# Funcion para actualizar el color de la pieza
def actualizar_color(step_index, total_steps):
    factor = step_index / (total_steps - 1)
    rojo  = color_inicial[0] + (color_final[0] - color_inicial[0]) * factor
    verde = color_inicial[1] + (color_final[1] - color_inicial[1]) * factor
    azul  = color_inicial[2] + (color_final[2] - color_inicial[2]) * factor
    obj.setColor([rojo, verde, azul, 1.0])

for target_name in targets:
    target = RDK.Item(target_name, ITEM_TYPE_TARGET)
    if not target.Valid():
        raise Exception(f'Target no encontrado: {target_name}')
    target_poses.append(target.Pose())

total_steps = len(target_poses)

# Ir a posición de inicio
home_joints = robot.JointsHome()
robot.MoveJ(home_joints)
robot.MoveJ(target_poses[0])

RDK.Spray_SetState(SPRAY_ON)

# Pintado con cambio progresivo de color (10 pasos)
for i, pose in enumerate(target_poses[1:10]):

    actualizar_color(step_index, total_steps)
    robot.MoveL(pose)
    step_index += 1

# Últimos movimientos
robot.setSpeed(50, 50)
robot.setAcceleration(50)
actualizar_color(step_index, total_steps)
robot.MoveL(target_poses[10])
step_index += 1
actualizar_color(step_index, total_steps)
robot.MoveL(target_poses[11])
step_index += 1

robot.setSpeed(10, 10)
robot.setAcceleration(10)
for pose in target_poses[12:15]:
    actualizar_color(step_index, total_steps)
    robot.MoveJ(pose)
    step_index += 1

# Bucle: 18 pasos de 5 grados
for i in range(18):
    # Obtener la pose actual en cada iteración (actualizada)
    pose_actual6 = frame6.Pose()
    pose_actual5 = frame5.Pose()

    # Crear una rotación de 5 grados en Z
    rot_5deg6 = robomath.rotz(math.radians(5))
    rot_5deg5 = robomath.rotz(math.radians(5))

    # Aplicar rotación acumulativa
    nueva_pose6 = pose_actual6 * rot_5deg6
    nueva_pose5 = pose_actual5 * rot_5deg5

    # Establecer la nueva pose
    frame6.setPose(nueva_pose6)
    frame5.setPose(nueva_pose5)

for pose in target_poses[15:29]:
    actualizar_color(step_index, total_steps)
    robot.MoveJ(pose)
    step_index += 1

robot.MoveJ(home_joints)

for pose in target_poses[30:33]:
    actualizar_color(step_index, total_steps)
    robot.MoveJ(pose)
    step_index += 1

# Bucle: 18 pasos de 5 grados
for i in range(18):
    # Obtener la pose actual en cada iteración (actualizada)
    pose_actual6 = frame6.Pose()
    pose_actual5 = frame5.Pose()

    # Crear una rotación de 5 grados en Z
    rot_5deg6 = robomath.rotz(math.radians(5))
    rot_5deg5 = robomath.rotz(math.radians(5))

    # Aplicar rotación acumulativa
    nueva_pose6 = pose_actual6 * rot_5deg6
    nueva_pose5 = pose_actual5 * rot_5deg5

    # Establecer la nueva pose
    frame6.setPose(nueva_pose6)
    frame5.setPose(nueva_pose5)

for pose in target_poses[33:47]:
    actualizar_color(step_index, total_steps)
    robot.MoveJ(pose)
    step_index += 1

# Bucle: 18 pasos de 5 grados
for i in range(18):
    # Obtener la pose actual en cada iteración (actualizada)
    pose_actual6 = frame6.Pose()
    pose_actual5 = frame5.Pose()

    # Crear una rotación de 5 grados en Z
    rot_5deg6 = robomath.rotz(math.radians(5))
    rot_5deg5 = robomath.rotz(math.radians(5))

    # Aplicar rotación acumulativa
    nueva_pose6 = pose_actual6 * rot_5deg6
    nueva_pose5 = pose_actual5 * rot_5deg5

    # Establecer la nueva pose
    frame6.setPose(nueva_pose6)
    frame5.setPose(nueva_pose5)

for pose in target_poses[47:]:
    actualizar_color(step_index, total_steps)
    robot.MoveJ(pose)
    step_index += 1

# Bucle: 18 pasos de 5 grados
for i in range(18):
    # Obtener la pose actual en cada iteración (actualizada)
    pose_actual6 = frame6.Pose()
    pose_actual5 = frame5.Pose()

    # Crear una rotación de 5 grados en Z
    rot_5deg6 = robomath.rotz(math.radians(5))
    rot_5deg5 = robomath.rotz(math.radians(5))

    # Aplicar rotación acumulativa
    nueva_pose6 = pose_actual6 * rot_5deg6
    nueva_pose5 = pose_actual5 * rot_5deg5

    # Establecer la nueva pose
    frame6.setPose(nueva_pose6)
    frame5.setPose(nueva_pose5)

robot.MoveJ(home_joints)
time.sleep(5.0)

robot.MoveJ(home_joints)
robot.MoveJ(target_poses[0])

RDK.Spray_SetState(SPRAY_ON)

# Pintado con cambio progresivo de color (10 pasos)
for i, pose in enumerate(target_poses[1:10]):

    actualizar_color(step_index, total_steps)
    robot.MoveL(pose)
    step_index += 1

# Últimos movimientos
robot.setSpeed(50, 50)
robot.setAcceleration(50)
actualizar_color(step_index, total_steps)
robot.MoveL(target_poses[10])
step_index += 1
actualizar_color(step_index, total_steps)
robot.MoveL(target_poses[11])
step_index += 1

robot.setSpeed(10, 10)
robot.setAcceleration(10)
for pose in target_poses[12:15]:
    actualizar_color(step_index, total_steps)
    robot.MoveJ(pose)
    step_index += 1

# Bucle: 18 pasos de 5 grados
for i in range(18):
    # Obtener la pose actual en cada iteración (actualizada)
    pose_actual6 = frame6.Pose()
    pose_actual5 = frame5.Pose()

    # Crear una rotación de 5 grados en Z
    rot_5deg6 = robomath.rotz(math.radians(5))
    rot_5deg5 = robomath.rotz(math.radians(5))

    # Aplicar rotación acumulativa
    nueva_pose6 = pose_actual6 * rot_5deg6
    nueva_pose5 = pose_actual5 * rot_5deg5

    # Establecer la nueva pose
    frame6.setPose(nueva_pose6)
    frame5.setPose(nueva_pose5)

for pose in target_poses[15:29]:
    actualizar_color(step_index, total_steps)
    robot.MoveJ(pose)
    step_index += 1

robot.MoveJ(home_joints)

for pose in target_poses[30:33]:
    actualizar_color(step_index, total_steps)
    robot.MoveJ(pose)
    step_index += 1

# Bucle: 18 pasos de 5 grados
for i in range(18):
    # Obtener la pose actual en cada iteración (actualizada)
    pose_actual6 = frame6.Pose()
    pose_actual5 = frame5.Pose()

    # Crear una rotación de 5 grados en Z
    rot_5deg6 = robomath.rotz(math.radians(5))
    rot_5deg5 = robomath.rotz(math.radians(5))

    # Aplicar rotación acumulativa
    nueva_pose6 = pose_actual6 * rot_5deg6
    nueva_pose5 = pose_actual5 * rot_5deg5

    # Establecer la nueva pose
    frame6.setPose(nueva_pose6)
    frame5.setPose(nueva_pose5)

for pose in target_poses[33:47]:
    actualizar_color(step_index, total_steps)
    robot.MoveJ(pose)
    step_index += 1

# Bucle: 18 pasos de 5 grados
for i in range(18):
    # Obtener la pose actual en cada iteración (actualizada)
    pose_actual6 = frame6.Pose()
    pose_actual5 = frame5.Pose()

    # Crear una rotación de 5 grados en Z
    rot_5deg6 = robomath.rotz(math.radians(5))
    rot_5deg5 = robomath.rotz(math.radians(5))

    # Aplicar rotación acumulativa
    nueva_pose6 = pose_actual6 * rot_5deg6
    nueva_pose5 = pose_actual5 * rot_5deg5

    # Establecer la nueva pose
    frame6.setPose(nueva_pose6)
    frame5.setPose(nueva_pose5)

for pose in target_poses[47:]:
    actualizar_color(step_index, total_steps)
    robot.MoveJ(pose)
    step_index += 1

# Bucle: 18 pasos de 5 grados
for i in range(18):
    # Obtener la pose actual en cada iteración (actualizada)
    pose_actual6 = frame6.Pose()
    pose_actual5 = frame5.Pose()

    # Crear una rotación de 5 grados en Z
    rot_5deg6 = robomath.rotz(math.radians(5))
    rot_5deg5 = robomath.rotz(math.radians(5))

    # Aplicar rotación acumulativa
    nueva_pose6 = pose_actual6 * rot_5deg6
    nueva_pose5 = pose_actual5 * rot_5deg5

    # Establecer la nueva pose
    frame6.setPose(nueva_pose6)
    frame5.setPose(nueva_pose5)

# Desactivar pintado al finalizar
RDK.Spray_Clear()
RDK.Spray_SetState(SPRAY_OFF)

--- Python program Chopper21 ---
from robodk.robolink import *  # API de RoboDK
from robodk.robomath import *  # Funciones matemáticas
import time
import math

# Inicializar conexión con RoboDK
RDK = Robolink()

# Borrar las partículas de pintura previas
RDK.Spray_Clear()

# Comprobar si estamos en modo simulación
if RDK.RunMode() != RUNMODE_SIMULATE:
    raise Exception('El robot no está en modo simulación')

# Obtener el robot
robot = RDK.Item('ABB IRB 580/12S 2', ITEM_TYPE_ROBOT)
if not robot.Valid():
    raise Exception('Robot "ABB IRB 580/12S 2" no encontrado')

# Establecer herramienta activa (TCP2)
tool = RDK.Item('TCP2', ITEM_TYPE_TOOL)
if not tool.Valid():
    raise Exception('Herramienta TCP2 no encontrada')
robot.setTool(tool)

# Obtener el objeto a pintar
obj = RDK.Item('Chopper Frame AP203 1', ITEM_TYPE_OBJECT)
if not obj.Valid():
    raise Exception('Objeto "Chopper Frame AP203 1" no encontrado')

# Obtener el sistema del gancho
frame6 = RDK.Item('Frame C1', ITEM_TYPE_FRAME)
if not frame6.Valid():
    raise Exception('Sistema "Frame C1" no encontrado')

# Obtener el sistema del objeto
frame4 = RDK.Item('Frame 4', ITEM_TYPE_FRAME)
if not frame4.Valid():
    raise Exception('Sistema "Frame 4" no encontrado')

# -------------------------
# MAPEO DE COLORES
# -------------------------
colores_numericos = {
    0: [1.0, 0.0, 0.0],  # rojo
    1: [0.0, 0.0, 0.0],  # negro
    2: [0.0, 1.0, 0.0],  # verde
    3: [0.5, 0.5, 0.5],  # gris
    4: [1.0, 1.0, 1.0],  # blanco
    5: [1.0, 0.5, 0.0]   # naranja
}

# Obtener número desde variable global de RoboDK
valor_color = RDK.getParam('ColorElegido2')
if valor_color is None:
    valor_color = 0  # valor por defecto
valor_color = int(valor_color)

if valor_color not in colores_numericos:
    raise Exception(f'ColorElegido inválido: {valor_color}')
color_final = colores_numericos[valor_color]

# Color neutro inicial
color_inicial = [0.9, 0.9, 0.9]

# Activar pintado automático
options_command = "ELLYPSE PROJECT PARTICLE=SPHERE(4,10,1,1,0.5) STEP=3x3 RAND=2"
close_param = [0, 0, 0, 5, 0, 0, 0, 5, 0, color_final[0], color_final[1], color_final[2], 1]
far_param   = [0, 0, 2000, 500, 0, 2000, 0, 500, 2000, color_final[0], color_final[1], color_final[2], 0.2]
volume = Mat([close_param, far_param]).tr()
RDK.Spray_Add(tool, obj, options_command, volume)
RDK.Spray_SetState(SPRAY_ON)

# Establecer velocidades lentas
robot.setSpeed(50, 50)
robot.setAcceleration(50)

# Lista de nombres de targets
targets = [
    'Pintura21_1',
    'Pintura21_2',
    'Pintura21_3',
    'Pintura21_4',
    'Pintura21_5',
    'Pintura21_6',
    'Pintura21_7',
    'Pintura21_8',
    'Pintura21_9',
    'Pintura21_8',
    'Pintura21_1',

    'Pintura21_11',
    'Pintura21_13',
    'Pintura21_14',
    'Pintura21_15',
    'Pintura21_16',
    'Pintura21_17',
    'Pintura21_18',
    'Pintura21_19',
    'Pintura21_13',
    'Pintura21_20',
    'Pintura21_1',

    'Pintura21_21',
    'Pintura21_22',
    'Pintura21_23',
    'Pintura21_24',
    'Pintura21_25',
    'Pintura21_26',
    'Pintura21_27',
    'Pintura21_28',
    'Pintura21_29',
    'Pintura21_28',
    'Pintura21_1',

    'Pintura21_31',
    'Pintura21_32',
    'Pintura21_39',
    'Pintura21_32',
    'Pintura21_33',
    'Pintura21_38',
    'Pintura21_34',
    'Pintura21_37',
    'Pintura21_35',
    'Pintura21_36',
    'Pintura21_37',
    'Pintura21_38',
    'Pintura21_39',
    'Pintura21_40'


]

# Obtener poses de targets
target_poses = []

# Contar los pasos totales en todas las fases

step_index = 0

# Funcion para actualizar el color de la pieza
def actualizar_color(step_index, total_steps):
    factor = step_index / (total_steps - 1)
    rojo  = color_inicial[0] + (color_final[0] - color_inicial[0]) * factor
    verde = color_inicial[1] + (color_final[1] - color_inicial[1]) * factor
    azul  = color_inicial[2] + (color_final[2] - color_inicial[2]) * factor
    obj.setColor([rojo, verde, azul, 1.0])

for target_name in targets:
    target = RDK.Item(target_name, ITEM_TYPE_TARGET)
    if not target.Valid():
        raise Exception(f'Target no encontrado: {target_name}')
    target_poses.append(target.Pose())

total_steps = len(target_poses)

# Ir a posición de inicio
home_joints = robot.JointsHome()
robot.MoveJ(home_joints)
robot.MoveJ(target_poses[0])

RDK.Spray_SetState(SPRAY_ON)

robot.setSpeed(10, 10)
robot.setAcceleration(10)

# Pintado con cambio progresivo de color (10 pasos)
for i, pose in enumerate(target_poses[1:10]):

    actualizar_color(step_index, total_steps)
    robot.MoveJ(pose)
    step_index += 1

# Últimos movimientos

robot.setSpeed(50, 50)
robot.setAcceleration(50)

actualizar_color(step_index, total_steps)
robot.MoveL(target_poses[11])
step_index += 1

# Bucle: 18 pasos de 5 grados
for i in range(18):
    # Obtener la pose actual en cada iteración (actualizada)
    pose_actual6 = frame6.Pose()
    pose_actual5 = frame4.Pose()

    # Crear una rotación de 5 grados en Z
    rot_5deg6 = robomath.rotz(math.radians(5))
    rot_5deg5 = robomath.rotz(math.radians(5))

    # Aplicar rotación acumulativa
    nueva_pose6 = pose_actual6 * rot_5deg6
    nueva_pose5 = pose_actual5 * rot_5deg5

    # Establecer la nueva pose
    frame6.setPose(nueva_pose6)
    frame4.setPose(nueva_pose5)

robot.setSpeed(10, 10)
robot.setAcceleration(10)

for pose in target_poses[12:23]:
    actualizar_color(step_index, total_steps)
    robot.MoveJ(pose)
    step_index += 1

# Bucle: 18 pasos de 5 grados
for i in range(18):
    # Obtener la pose actual en cada iteración (actualizada)
    pose_actual6 = frame6.Pose()
    pose_actual5 = frame4.Pose()

    # Crear una rotación de 5 grados en Z
    rot_5deg6 = robomath.rotz(math.radians(5))
    rot_5deg5 = robomath.rotz(math.radians(5))

    # Aplicar rotación acumulativa
    nueva_pose6 = pose_actual6 * rot_5deg6
    nueva_pose5 = pose_actual5 * rot_5deg5

    # Establecer la nueva pose
    frame6.setPose(nueva_pose6)
    frame4.setPose(nueva_pose5)

for pose in target_poses[23:33]:
    actualizar_color(step_index, total_steps)
    robot.MoveJ(pose)
    step_index += 1

robot.MoveJ(home_joints)

# Bucle: 18 pasos de 5 grados
for i in range(18):
    # Obtener la pose actual en cada iteración (actualizada)
    pose_actual6 = frame6.Pose()
    pose_actual5 = frame4.Pose()

    # Crear una rotación de 5 grados en Z
    rot_5deg6 = robomath.rotz(math.radians(5))
    rot_5deg5 = robomath.rotz(math.radians(5))

    # Aplicar rotación acumulativa
    nueva_pose6 = pose_actual6 * rot_5deg6
    nueva_pose5 = pose_actual5 * rot_5deg5

    # Establecer la nueva pose
    frame6.setPose(nueva_pose6)
    frame4.setPose(nueva_pose5)

for pose in target_poses[33:]:
    actualizar_color(step_index, total_steps)
    robot.MoveJ(pose)
    step_index += 1

robot.MoveJ(home_joints)

# Bucle: 18 pasos de 5 grados
for i in range(18):
    # Obtener la pose actual en cada iteración (actualizada)
    pose_actual6 = frame6.Pose()
    pose_actual5 = frame4.Pose()

    # Crear una rotación de 5 grados en Z
    rot_5deg6 = robomath.rotz(math.radians(5))
    rot_5deg5 = robomath.rotz(math.radians(5))

    # Aplicar rotación acumulativa
    nueva_pose6 = pose_actual6 * rot_5deg6
    nueva_pose5 = pose_actual5 * rot_5deg5

    # Establecer la nueva pose
    frame6.setPose(nueva_pose6)
    frame4.setPose(nueva_pose5)

robot.MoveJ(home_joints)
time.sleep(5.0)

robot.MoveJ(home_joints)
robot.MoveJ(target_poses[0])

RDK.Spray_SetState(SPRAY_ON)

robot.setSpeed(10, 10)
robot.setAcceleration(10)

# Pintado con cambio progresivo de color (10 pasos)
for i, pose in enumerate(target_poses[1:10]):

    actualizar_color(step_index, total_steps)
    robot.MoveJ(pose)
    step_index += 1

# Últimos movimientos

robot.setSpeed(50, 50)
robot.setAcceleration(50)

actualizar_color(step_index, total_steps)
robot.MoveL(target_poses[11])
step_index += 1

# Bucle: 18 pasos de 5 grados
for i in range(18):
    # Obtener la pose actual en cada iteración (actualizada)
    pose_actual6 = frame6.Pose()
    pose_actual5 = frame4.Pose()

    # Crear una rotación de 5 grados en Z
    rot_5deg6 = robomath.rotz(math.radians(5))
    rot_5deg5 = robomath.rotz(math.radians(5))

    # Aplicar rotación acumulativa
    nueva_pose6 = pose_actual6 * rot_5deg6
    nueva_pose5 = pose_actual5 * rot_5deg5

    # Establecer la nueva pose
    frame6.setPose(nueva_pose6)
    frame4.setPose(nueva_pose5)

robot.setSpeed(10, 10)
robot.setAcceleration(10)

for pose in target_poses[12:23]:
    actualizar_color(step_index, total_steps)
    robot.MoveJ(pose)
    step_index += 1

# Bucle: 18 pasos de 5 grados
for i in range(18):
    # Obtener la pose actual en cada iteración (actualizada)
    pose_actual6 = frame6.Pose()
    pose_actual5 = frame4.Pose()

    # Crear una rotación de 5 grados en Z
    rot_5deg6 = robomath.rotz(math.radians(5))
    rot_5deg5 = robomath.rotz(math.radians(5))

    # Aplicar rotación acumulativa
    nueva_pose6 = pose_actual6 * rot_5deg6
    nueva_pose5 = pose_actual5 * rot_5deg5

    # Establecer la nueva pose
    frame6.setPose(nueva_pose6)
    frame4.setPose(nueva_pose5)

for pose in target_poses[23:33]:
    actualizar_color(step_index, total_steps)
    robot.MoveJ(pose)
    step_index += 1

robot.MoveJ(home_joints)

# Bucle: 18 pasos de 5 grados
for i in range(18):
    # Obtener la pose actual en cada iteración (actualizada)
    pose_actual6 = frame6.Pose()
    pose_actual5 = frame4.Pose()

    # Crear una rotación de 5 grados en Z
    rot_5deg6 = robomath.rotz(math.radians(5))
    rot_5deg5 = robomath.rotz(math.radians(5))

    # Aplicar rotación acumulativa
    nueva_pose6 = pose_actual6 * rot_5deg6
    nueva_pose5 = pose_actual5 * rot_5deg5

    # Establecer la nueva pose
    frame6.setPose(nueva_pose6)
    frame4.setPose(nueva_pose5)

for pose in target_poses[33:]:
    actualizar_color(step_index, total_steps)
    robot.MoveJ(pose)
    step_index += 1

robot.MoveJ(home_joints)

# Bucle: 18 pasos de 5 grados
for i in range(18):
    # Obtener la pose actual en cada iteración (actualizada)
    pose_actual6 = frame6.Pose()
    pose_actual5 = frame4.Pose()

    # Crear una rotación de 5 grados en Z
    rot_5deg6 = robomath.rotz(math.radians(5))
    rot_5deg5 = robomath.rotz(math.radians(5))

    # Aplicar rotación acumulativa
    nueva_pose6 = pose_actual6 * rot_5deg6
    nueva_pose5 = pose_actual5 * rot_5deg5

    # Establecer la nueva pose
    frame6.setPose(nueva_pose6)
    frame4.setPose(nueva_pose5)

# Desactivar pintado al finalizar
RDK.Spray_Clear()
RDK.Spray_SetState(SPRAY_OFF)

--- Python program Chopper22 ---
from robodk.robolink import *  # API de RoboDK
from robodk.robomath import *  # Funciones matemáticas
import time
import math

# Inicializar conexión con RoboDK
RDK = Robolink()

# Borrar las partículas de pintura previas
RDK.Spray_Clear()

# Comprobar si estamos en modo simulación
if RDK.RunMode() != RUNMODE_SIMULATE:
    raise Exception('El robot no está en modo simulación')

# Obtener el robot
robot = RDK.Item('ABB IRB 580/12S 2', ITEM_TYPE_ROBOT)
if not robot.Valid():
    raise Exception('Robot "ABB IRB 580/12S 2" no encontrado')

# Establecer herramienta activa (TCP2)
tool = RDK.Item('TCP2', ITEM_TYPE_TOOL)
if not tool.Valid():
    raise Exception('Herramienta TCP2 no encontrada')
robot.setTool(tool)

# Obtener el objeto a pintar
obj = RDK.Item('Chopper Frame AP203 2', ITEM_TYPE_OBJECT)
if not obj.Valid():
    raise Exception('Objeto "Chopper Frame AP203 2" no encontrado')

# Obtener el sistema del gancho
frame6 = RDK.Item('Frame C2', ITEM_TYPE_FRAME)
if not frame6.Valid():
    raise Exception('Sistema "Frame C2" no encontrado')

# Obtener el sistema del objeto
frame4 = RDK.Item('Frame 6', ITEM_TYPE_FRAME)
if not frame4.Valid():
    raise Exception('Sistema "Frame 6" no encontrado')

# -------------------------
# MAPEO DE COLORES
# -------------------------
colores_numericos = {
    0: [1.0, 0.0, 0.0],  # rojo
    1: [0.0, 0.0, 0.0],  # negro
    2: [0.0, 1.0, 0.0],  # verde
    3: [0.5, 0.5, 0.5],  # gris
    4: [1.0, 1.0, 1.0],  # blanco
    5: [1.0, 0.5, 0.0]   # naranja
}

# Obtener número desde variable global de RoboDK
valor_color = RDK.getParam('ColorElegido2')
if valor_color is None:
    valor_color = 0  # valor por defecto
valor_color = int(valor_color)

if valor_color not in colores_numericos:
    raise Exception(f'ColorElegido inválido: {valor_color}')
color_final = colores_numericos[valor_color]

# Color neutro inicial
color_inicial = [0.9, 0.9, 0.9]

# Activar pintado automático
options_command = "ELLYPSE PROJECT PARTICLE=SPHERE(4,10,1,1,0.5) STEP=3x3 RAND=2"
close_param = [0, 0, 0, 5, 0, 0, 0, 5, 0, color_final[0], color_final[1], color_final[2], 1]
far_param   = [0, 0, 2000, 500, 0, 2000, 0, 500, 2000, color_final[0], color_final[1], color_final[2], 0.2]
volume = Mat([close_param, far_param]).tr()
RDK.Spray_Add(tool, obj, options_command, volume)
RDK.Spray_SetState(SPRAY_ON)

# Establecer velocidades lentas
robot.setSpeed(50, 50)
robot.setAcceleration(50)

# Lista de nombres de targets
targets = [
    'Pintura21_1',
    'Pintura21_2',
    'Pintura21_3',
    'Pintura21_4',
    'Pintura21_5',
    'Pintura21_6',
    'Pintura21_7',
    'Pintura21_8',
    'Pintura21_9',
    'Pintura21_8',
    'Pintura21_1',

    'Pintura21_11',
    'Pintura21_13',
    'Pintura21_14',
    'Pintura21_15',
    'Pintura21_16',
    'Pintura21_17',
    'Pintura21_18',
    'Pintura21_19',
    'Pintura21_13',
    'Pintura21_20',
    'Pintura21_1',

    'Pintura21_21',
    'Pintura21_22',
    'Pintura21_23',
    'Pintura21_24',
    'Pintura21_25',
    'Pintura21_26',
    'Pintura21_27',
    'Pintura21_28',
    'Pintura21_29',
    'Pintura21_28',
    'Pintura21_1',

    'Pintura21_31',
    'Pintura21_32',
    'Pintura21_39',
    'Pintura21_32',
    'Pintura21_33',
    'Pintura21_38',
    'Pintura21_34',
    'Pintura21_37',
    'Pintura21_35',
    'Pintura21_36',
    'Pintura21_37',
    'Pintura21_38',
    'Pintura21_39',
    'Pintura21_40'


]

# Obtener poses de targets
target_poses = []

# Contar los pasos totales en todas las fases

step_index = 0

# Funcion para actualizar el color de la pieza
def actualizar_color(step_index, total_steps):
    factor = step_index / (total_steps - 1)
    rojo  = color_inicial[0] + (color_final[0] - color_inicial[0]) * factor
    verde = color_inicial[1] + (color_final[1] - color_inicial[1]) * factor
    azul  = color_inicial[2] + (color_final[2] - color_inicial[2]) * factor
    obj.setColor([rojo, verde, azul, 1.0])

for target_name in targets:
    target = RDK.Item(target_name, ITEM_TYPE_TARGET)
    if not target.Valid():
        raise Exception(f'Target no encontrado: {target_name}')
    target_poses.append(target.Pose())

total_steps = len(target_poses)

# Ir a posición de inicio
home_joints = robot.JointsHome()
robot.MoveJ(home_joints)
robot.MoveJ(target_poses[0])

RDK.Spray_SetState(SPRAY_ON)

robot.setSpeed(10, 10)
robot.setAcceleration(10)

# Pintado con cambio progresivo de color (10 pasos)
for i, pose in enumerate(target_poses[1:10]):

    actualizar_color(step_index, total_steps)
    robot.MoveJ(pose)
    step_index += 1

# Últimos movimientos

robot.setSpeed(50, 50)
robot.setAcceleration(50)

actualizar_color(step_index, total_steps)
robot.MoveL(target_poses[11])
step_index += 1

# Bucle: 18 pasos de 5 grados
for i in range(18):
    # Obtener la pose actual en cada iteración (actualizada)
    pose_actual6 = frame6.Pose()
    pose_actual5 = frame4.Pose()

    # Crear una rotación de 5 grados en Z
    rot_5deg6 = robomath.rotz(math.radians(5))
    rot_5deg5 = robomath.rotz(math.radians(5))

    # Aplicar rotación acumulativa
    nueva_pose6 = pose_actual6 * rot_5deg6
    nueva_pose5 = pose_actual5 * rot_5deg5

    # Establecer la nueva pose
    frame6.setPose(nueva_pose6)
    frame4.setPose(nueva_pose5)

robot.setSpeed(10, 10)
robot.setAcceleration(10)

for pose in target_poses[12:23]:
    actualizar_color(step_index, total_steps)
    robot.MoveJ(pose)
    step_index += 1

# Bucle: 18 pasos de 5 grados
for i in range(18):
    # Obtener la pose actual en cada iteración (actualizada)
    pose_actual6 = frame6.Pose()
    pose_actual5 = frame4.Pose()

    # Crear una rotación de 5 grados en Z
    rot_5deg6 = robomath.rotz(math.radians(5))
    rot_5deg5 = robomath.rotz(math.radians(5))

    # Aplicar rotación acumulativa
    nueva_pose6 = pose_actual6 * rot_5deg6
    nueva_pose5 = pose_actual5 * rot_5deg5

    # Establecer la nueva pose
    frame6.setPose(nueva_pose6)
    frame4.setPose(nueva_pose5)

for pose in target_poses[23:33]:
    actualizar_color(step_index, total_steps)
    robot.MoveJ(pose)
    step_index += 1

robot.MoveJ(home_joints)

# Bucle: 18 pasos de 5 grados
for i in range(18):
    # Obtener la pose actual en cada iteración (actualizada)
    pose_actual6 = frame6.Pose()
    pose_actual5 = frame4.Pose()

    # Crear una rotación de 5 grados en Z
    rot_5deg6 = robomath.rotz(math.radians(5))
    rot_5deg5 = robomath.rotz(math.radians(5))

    # Aplicar rotación acumulativa
    nueva_pose6 = pose_actual6 * rot_5deg6
    nueva_pose5 = pose_actual5 * rot_5deg5

    # Establecer la nueva pose
    frame6.setPose(nueva_pose6)
    frame4.setPose(nueva_pose5)

for pose in target_poses[33:]:
    actualizar_color(step_index, total_steps)
    robot.MoveJ(pose)
    step_index += 1

robot.MoveJ(home_joints)

# Bucle: 18 pasos de 5 grados
for i in range(18):
    # Obtener la pose actual en cada iteración (actualizada)
    pose_actual6 = frame6.Pose()
    pose_actual5 = frame4.Pose()

    # Crear una rotación de 5 grados en Z
    rot_5deg6 = robomath.rotz(math.radians(5))
    rot_5deg5 = robomath.rotz(math.radians(5))

    # Aplicar rotación acumulativa
    nueva_pose6 = pose_actual6 * rot_5deg6
    nueva_pose5 = pose_actual5 * rot_5deg5

    # Establecer la nueva pose
    frame6.setPose(nueva_pose6)
    frame4.setPose(nueva_pose5)

robot.MoveJ(home_joints)
time.sleep(5.0)

robot.MoveJ(home_joints)
robot.MoveJ(target_poses[0])

RDK.Spray_SetState(SPRAY_ON)

robot.setSpeed(10, 10)
robot.setAcceleration(10)

# Pintado con cambio progresivo de color (10 pasos)
for i, pose in enumerate(target_poses[1:10]):

    actualizar_color(step_index, total_steps)
    robot.MoveJ(pose)
    step_index += 1

# Últimos movimientos

robot.setSpeed(50, 50)
robot.setAcceleration(50)

actualizar_color(step_index, total_steps)
robot.MoveL(target_poses[11])
step_index += 1

# Bucle: 18 pasos de 5 grados
for i in range(18):
    # Obtener la pose actual en cada iteración (actualizada)
    pose_actual6 = frame6.Pose()
    pose_actual5 = frame4.Pose()

    # Crear una rotación de 5 grados en Z
    rot_5deg6 = robomath.rotz(math.radians(5))
    rot_5deg5 = robomath.rotz(math.radians(5))

    # Aplicar rotación acumulativa
    nueva_pose6 = pose_actual6 * rot_5deg6
    nueva_pose5 = pose_actual5 * rot_5deg5

    # Establecer la nueva pose
    frame6.setPose(nueva_pose6)
    frame4.setPose(nueva_pose5)

robot.setSpeed(10, 10)
robot.setAcceleration(10)

for pose in target_poses[12:23]:
    actualizar_color(step_index, total_steps)
    robot.MoveJ(pose)
    step_index += 1

# Bucle: 18 pasos de 5 grados
for i in range(18):
    # Obtener la pose actual en cada iteración (actualizada)
    pose_actual6 = frame6.Pose()
    pose_actual5 = frame4.Pose()

    # Crear una rotación de 5 grados en Z
    rot_5deg6 = robomath.rotz(math.radians(5))
    rot_5deg5 = robomath.rotz(math.radians(5))

    # Aplicar rotación acumulativa
    nueva_pose6 = pose_actual6 * rot_5deg6
    nueva_pose5 = pose_actual5 * rot_5deg5

    # Establecer la nueva pose
    frame6.setPose(nueva_pose6)
    frame4.setPose(nueva_pose5)

for pose in target_poses[23:33]:
    actualizar_color(step_index, total_steps)
    robot.MoveJ(pose)
    step_index += 1

robot.MoveJ(home_joints)

# Bucle: 18 pasos de 5 grados
for i in range(18):
    # Obtener la pose actual en cada iteración (actualizada)
    pose_actual6 = frame6.Pose()
    pose_actual5 = frame4.Pose()

    # Crear una rotación de 5 grados en Z
    rot_5deg6 = robomath.rotz(math.radians(5))
    rot_5deg5 = robomath.rotz(math.radians(5))

    # Aplicar rotación acumulativa
    nueva_pose6 = pose_actual6 * rot_5deg6
    nueva_pose5 = pose_actual5 * rot_5deg5

    # Establecer la nueva pose
    frame6.setPose(nueva_pose6)
    frame4.setPose(nueva_pose5)

for pose in target_poses[33:]:
    actualizar_color(step_index, total_steps)
    robot.MoveJ(pose)
    step_index += 1

robot.MoveJ(home_joints)

# Bucle: 18 pasos de 5 grados
for i in range(18):
    # Obtener la pose actual en cada iteración (actualizada)
    pose_actual6 = frame6.Pose()
    pose_actual5 = frame4.Pose()

    # Crear una rotación de 5 grados en Z
    rot_5deg6 = robomath.rotz(math.radians(5))
    rot_5deg5 = robomath.rotz(math.radians(5))

    # Aplicar rotación acumulativa
    nueva_pose6 = pose_actual6 * rot_5deg6
    nueva_pose5 = pose_actual5 * rot_5deg5

    # Establecer la nueva pose
    frame6.setPose(nueva_pose6)
    frame4.setPose(nueva_pose5)

# Desactivar pintado al finalizar
RDK.Spray_Clear()
RDK.Spray_SetState(SPRAY_OFF)

--- Python program SprayOn ---
# This macro allows simulating a spray gun for painting or to simulate the trace of inspaction
#
# You can call SprayOn(1) to simulate turning the Spray gun ON or SprayOn(0) to stop simulating the gun
# Calling SprayOn(-1) clears all displayed data
# The macro will output spray gun statistics
#
# --------------------------------------------------------------
# This script shows how to create "spray" object in RoboDK that allows simulating particle deposition by using:
# RDK.Spray_Add(tool, object, options_command, volume, geometry)
#    tool: tool item (TCP) to use
#    object: object to project the particles
#    options_command (optional): string to specify options.
#    volume (optional): Matrix of parameters defining the volume of the spray gun
#    geometry (optional): Matrix of vertices defining the triangles.
#
# More information here:
# https://robodk.com/doc/en/PythonAPI/robodk.html#robodk.robolink.Robolink.Spray_Add
# https://robodk.com/doc/en/RoboDK-API.html
#
# The scripts ArcStart, ArcEnd and WeldOn and SpindleOn behave in a similar way, the only difference is the default behavior
# This behavior simmulates Fanuc Arc Welding and triggers appropriate output when using the customized post processor.
# Select ESC to clear the trace manually.
#
# Example scripts that use Spray_Add:
#     SpindleOn / SpindleOff    -> Turn trace On/Off
#     ArcOn / ArcOff            -> Turn trace On/Off
#     SprayOn / SprayOff        -> Simulate a spray given a workspace volume (for painting)
#     WeldOn / WeldOff          -> Support for multiple weld guns

#------------------------------------------------------------------

# Use a specific tool as a spray gun
Tool_Name = 'TCP1'
#Tool_Name = 'Tool 2'

# Use a specific object to project particles:
Object_Name = 'Frame cb 750'
#Object_Name = 'Part'

# Define the default action (0 to deactivate, +1 to activate, -1 to clear any spray gun simulation)
# Setting it to None will display a message
ACTION = None

from robodk.robolink import *  # API to communicate with RoboDK
from robodk.robomath import *  # basic matrix operations
from robodk.robodialogs import *

RDK = Robolink()

# quit if we are not in simulation mode
if RDK.RunMode() != RUNMODE_SIMULATE:
    quit()

# Get any previously added spray gun simulations and display statistics (spray on the part vs spray falling out of the part)
info, data = RDK.Spray_GetStats()
if data.size(1) > 0:
    print("Spray gun statistics:")
    print(info)
    print(data.tr())
    # # Diplay statistics
    # RDK.ShowMessage("Material used: %.1f%%<br>Material waisted: %.1f%%<br>Total particles: %.1f" % (data[1,0],data[2,0],data[3,0]), True)
    # # Clear previous spray
    # RDK.Spray_Clear()

# Check if we are running this program inside another program and passing arguments
import sys
if len(sys.argv) > 1:
    ACTION = int(sys.argv[1])

# If the default ACTION is None, display a message to activate/deactivate the spray gun
if ACTION is None:
    print('Note: This macro can be called as Spray(1) or SprayOn(0)')
    entry = mbox('Turn gun ON or OFF', ('On', '1'), ('Off', '0'))
    if not entry:
        quit()
    ACTION = int(entry)

if ACTION == 0:
    # Turn the gun off
    RDK.Spray_SetState(SPRAY_OFF)

elif ACTION < 0:
    # Clear all spray simulations (same as pressing ESC key)
    RDK.Spray_Clear()

elif ACTION > 0:
    # Create a new spray gun object in RoboDK
    # by using RDK.Spray_Add(tool, object, options_command, volume, geometry)
    # tool: tool item (TCP) to use
    # object: object to project the particles
    # options_command (optional): string to specify options. Example:
    #     STEP=AxB: Defines the grid to be projected 1x1 means only one line of particle projection (for example, for welding)
    #     PARTICLE: Defines the shape and size of particle (sphere or particle), unless a specific geometry is provided:
    #       a- SPHERE(radius, facets)
    #       b- SPHERE(radius, facets, scalex, scaley, scalez)
    #       b- CUBE(sizex, sizey, sizez)
    #     RAND=factor: Defines a random factor factor 0 means that the particles are not deposited randomly
    #     ELLYPSE: defines the volume as an ellypse (default)
    #     RECTANGLE: defines the volume as a rectangle
    #     PROJECT: project the particles to the surface (default) (for welding, painting or scanning)
    #     NO_PROJECT: does not project the particles to the surface (for example, for 3D printing)
    #
    # volume (optional): Matrix of parameters defining the volume of the spray gun
    # geometry (optional): Matrix of vertices defining the triangles.

    tool = 0  # auto detect active tool
    obj = 0  # auto detect object in active reference frame
    if Tool_Name is not None:
        tool = RDK.Item(Tool_Name, ITEM_TYPE_TOOL)

    if Object_Name is not None:
        obj = RDK.Item(Object_Name, ITEM_TYPE_OBJECT)
    # We can specify a given tool object and/or object
    #robot = RDK.Item("ABB IRB 2600-12/1.85", ITEM_TYPE_ROBOT)
    #tools = robot.Childs()
    #if len(tools) > 0:
    #    tool = tools[0]
    #obj = RDK.Item('object', ITEM_TYPE_OBJECT)

    options_command = "ELLYPSE PROJECT PARTICLE=SPHERE(4,8,1,1,0.5) STEP=6x6 RAND=2"  # simulate
    #options_command = "PARTICLE=CUBE(10,10,2) STEP=8x8"
    #options_command = "PARTICLE=SPHERE(4,8) STEP=8x8"
    #options_command = "PARTICLE=SPHERE(4,8,1,1,0.1) STEP=8x8 RAND=3"

    # Example commands for welding:
    # options_command = "PROJECT PARTICLE=SPHERE(4,8)"
    # options_command = PARTICLE=SPHERE(4,8) STEP=1x0

    # define the ellypse volume as p0, pA, pB, colorRGBA (close and far), in mm
    # coordinates must be provided with respect to the TCP
    close_p0 = [0, 0, 0]  # xyz in mm: Center of the conical ellypse (side 1)
    close_pA = [5, 0, 0]  # xyz in mm: First vertex of the conical ellypse (side 1)
    close_pB = [0, 5, 0]  # xyz in mm: Second vertex of the conical ellypse (side 1)
    close_color = [1, 0, 0, 1]  # RGBA (0-1)

    far_p0 = [0, 0, 2000]  # xyz in mm: Center of the conical ellypse (side 2)
    far_pA = [500, 0, 2000]  # xyz in mm: First vertex of the conical ellypse (side 2)
    far_pB = [0, 500, 2000]  # xyz in mm: Second vertex of the conical ellypse (side 2)
    far_color = [0, 0, 1, 0.2]  # RGBA (0-1)

    close_param = close_p0 + close_pA + close_pB + close_color
    far_param = far_p0 + far_pA + far_pB + far_color
    volume = Mat([close_param, far_param]).tr()
    RDK.Spray_Add(tool, obj, options_command, volume)
    RDK.Spray_SetState(SPRAY_ON)

    # Another example with a varying rectancular shape
    # define the rectangular volume as p0, pA, pB, colorRGBA (close and far)
    # close_param = [-90,-117,  0,  90,-117,0,   -90,117,  0,       0.2,0.2,1,.1]
    # far_param   = [-175,-190,200, 175,-190,200,   -175,190,200,   0.5,0,0,.9]
    # volume = Mat([close_param, far_param])
    # RDK.Spray_Add(tool, obj, "RECTANGLE PARTICLE=SPHERE(2,5) STEP=15x15 RAND=3", volume.tr())
    # RDK.Spray_SetState(SPRAY_ON)

    # Optional: define geometry as a list of triangles with normals (instead of a scaled cube or a sphere)
    # geom = Mat([[0,0,0,   0,0,1], [5,0,0,   0,0,1], [0,5,0,   0,0,1]])
    # RDK.Spray_Add(tool, obj, "STEP=8x8 RANDX=3", volume.tr(), geom.tr())
    # RDK.Spray_SetState(SPRAY_ON)

--- Python program MoverHonda11 ---
from robodk.robolink import *  # API de RoboDK
from robodk.robomath import *  # Funciones matemáticas
import time

# Inicializar conexión con RoboDK
RDK = Robolink()

# Obtener los frames
frame_H = RDK.Item('Frame H1', ITEM_TYPE_FRAME)
frame_5 = RDK.Item('Frame 5', ITEM_TYPE_FRAME)

if not frame_H.Valid() or not frame_5.Valid():
    raise Exception('Frames no válidos.')

# === Definir poses iniciales y finales manualmente ===

# Frame H
p_1_H = [448.718, 7875.499, 2280.872]
p_2_H = [448.718, 3935.499, 2280.872]
p_3_H = [2478.718, 1935.499, 2280.872]
p_4_H = [2478.718, 415.499, 2280.872]

# Frame 5
p_1_5 = [455.915, 7880.000, 1357.578]
p_2_5 = [455.915, 3940.000, 1357.578]
p_3_5 = [2485.915, 1940.000, 1357.578]
p_4_5 = [2485.915, 420.000, 1357.578]

# Número de pasos para la animación
pasos = 60
espera = 0.03

# Bucle de interpolación de p_1_H a p_2_H
for i in range(pasos + 1):
    t = i / pasos

    # Interpolar posición y rotación para Frame H
    px_H = p_1_H[0] + (p_2_H[0] - p_1_H[0]) * t
    py_H = p_1_H[1] + (p_2_H[1] - p_1_H[1]) * t
    pz_H = p_1_H[2] + (p_2_H[2] - p_1_H[2]) * t

    # Interpolar posición y rotación para Frame 5
    px_5 = p_1_5[0] + (p_2_5[0] - p_1_5[0]) * t
    py_5 = p_1_5[1] + (p_2_5[1] - p_1_5[1]) * t
    pz_5 = p_1_5[2] + (p_2_5[2] - p_1_5[2]) * t

    # Aplicar las nuevas poses
    frame_H.setPose(transl(px_H, py_H, pz_H))
    frame_5.setPose(transl(px_5, py_5, pz_5))

    time.sleep(espera)

# Bucle de interpolación de p_2_H a p_3_H
for i in range(pasos + 1):
    t = i / pasos

    # Interpolar posición y rotación para Frame H
    px_H = p_2_H[0] + (p_3_H[0] - p_2_H[0]) * t
    py_H = p_2_H[1] + (p_3_H[1] - p_2_H[1]) * t
    pz_H = p_2_H[2] + (p_3_H[2] - p_2_H[2]) * t

    # Interpolar posición y rotación para Frame 5
    px_5 = p_2_5[0] + (p_3_5[0] - p_2_5[0]) * t
    py_5 = p_2_5[1] + (p_3_5[1] - p_2_5[1]) * t
    pz_5 = p_2_5[2] + (p_3_5[2] - p_2_5[2]) * t

    # Aplicar las nuevas poses
    frame_H.setPose(transl(px_H, py_H, pz_H))
    frame_5.setPose(transl(px_5, py_5, pz_5))

    time.sleep(espera)

# Bucle de interpolación de p_3_H a p_4_H
for i in range(pasos + 1):
    t = i / pasos

    # Interpolar posición y rotación para Frame H
    px_H = p_3_H[0] + (p_4_H[0] - p_3_H[0]) * t
    py_H = p_3_H[1] + (p_4_H[1] - p_3_H[1]) * t
    pz_H = p_3_H[2] + (p_4_H[2] - p_3_H[2]) * t

    # Interpolar posición y rotación para Frame 5
    px_5 = p_3_5[0] + (p_4_5[0] - p_3_5[0]) * t
    py_5 = p_3_5[1] + (p_4_5[1] - p_3_5[1]) * t
    pz_5 = p_3_5[2] + (p_4_5[2] - p_3_5[2]) * t

    # Aplicar las nuevas poses
    frame_H.setPose(transl(px_H, py_H, pz_H))
    frame_5.setPose(transl(px_5, py_5, pz_5))

    time.sleep(espera)

--- Python program MoverHonda12 ---
from robodk.robolink import *  # API de RoboDK
from robodk.robomath import *  # Funciones matemáticas
import time

# Inicializar conexión con RoboDK
RDK = Robolink()

# Obtener los frames
frame_H = RDK.Item('Frame H2', ITEM_TYPE_FRAME)
frame_5 = RDK.Item('Frame 7', ITEM_TYPE_FRAME)

if not frame_H.Valid() or not frame_5.Valid():
    raise Exception('Frames no válidos.')

# === Definir poses iniciales y finales manualmente ===

# Frame H
p_1_H = [448.718, 7875.499, 2280.872]
p_2_H = [448.718, 3935.499, 2280.872]
p_3_H = [2478.718, 1935.499, 2280.872]
p_4_H = [2478.718, 415.499, 2280.872]

# Frame 5
p_1_5 = [455.915, 7880.000, 1357.578]
p_2_5 = [455.915, 3940.000, 1357.578]
p_3_5 = [2485.915, 1940.000, 1357.578]
p_4_5 = [2485.915, 420.000, 1357.578]

# Número de pasos para la animación
pasos = 60
espera = 0.03

# Bucle de interpolación de p_1_H a p_2_H
for i in range(pasos + 1):
    t = i / pasos

    # Interpolar posición y rotación para Frame H
    px_H = p_1_H[0] + (p_2_H[0] - p_1_H[0]) * t
    py_H = p_1_H[1] + (p_2_H[1] - p_1_H[1]) * t
    pz_H = p_1_H[2] + (p_2_H[2] - p_1_H[2]) * t

    # Interpolar posición y rotación para Frame 5
    px_5 = p_1_5[0] + (p_2_5[0] - p_1_5[0]) * t
    py_5 = p_1_5[1] + (p_2_5[1] - p_1_5[1]) * t
    pz_5 = p_1_5[2] + (p_2_5[2] - p_1_5[2]) * t

    # Aplicar las nuevas poses
    frame_H.setPose(transl(px_H, py_H, pz_H))
    frame_5.setPose(transl(px_5, py_5, pz_5))

    time.sleep(espera)

# Bucle de interpolación de p_2_H a p_3_H
for i in range(pasos + 1):
    t = i / pasos

    # Interpolar posición y rotación para Frame H
    px_H = p_2_H[0] + (p_3_H[0] - p_2_H[0]) * t
    py_H = p_2_H[1] + (p_3_H[1] - p_2_H[1]) * t
    pz_H = p_2_H[2] + (p_3_H[2] - p_2_H[2]) * t

    # Interpolar posición y rotación para Frame 5
    px_5 = p_2_5[0] + (p_3_5[0] - p_2_5[0]) * t
    py_5 = p_2_5[1] + (p_3_5[1] - p_2_5[1]) * t
    pz_5 = p_2_5[2] + (p_3_5[2] - p_2_5[2]) * t

    # Aplicar las nuevas poses
    frame_H.setPose(transl(px_H, py_H, pz_H))
    frame_5.setPose(transl(px_5, py_5, pz_5))

    time.sleep(espera)

# Bucle de interpolación de p_3_H a p_4_H
for i in range(pasos + 1):
    t = i / pasos

    # Interpolar posición y rotación para Frame H
    px_H = p_3_H[0] + (p_4_H[0] - p_3_H[0]) * t
    py_H = p_3_H[1] + (p_4_H[1] - p_3_H[1]) * t
    pz_H = p_3_H[2] + (p_4_H[2] - p_3_H[2]) * t

    # Interpolar posición y rotación para Frame 5
    px_5 = p_3_5[0] + (p_4_5[0] - p_3_5[0]) * t
    py_5 = p_3_5[1] + (p_4_5[1] - p_3_5[1]) * t
    pz_5 = p_3_5[2] + (p_4_5[2] - p_3_5[2]) * t

    # Aplicar las nuevas poses
    frame_H.setPose(transl(px_H, py_H, pz_H))
    frame_5.setPose(transl(px_5, py_5, pz_5))

    time.sleep(espera)

--- Python program MoverChopper11 ---
from robodk.robolink import *  # API de RoboDK
from robodk.robomath import *  # Funciones matemáticas
import time

# Inicializar conexión con RoboDK
RDK = Robolink()

# Obtener los frames
frame_C = RDK.Item('Frame C1', ITEM_TYPE_FRAME)
frame_4 = RDK.Item('Frame 4', ITEM_TYPE_FRAME)

if not frame_C.Valid() or not frame_4.Valid():
    raise Exception('Frames no válidos.')

# === Definir poses iniciales y finales manualmente ===

# Frame C
p_1_C = [4518.718, 7875.499, 2280.872]
p_2_C = [4518.718, 3935.499, 2280.872]
p_3_C = [2478.718, 1935.499, 2280.872]
p_4_C = [2478.718, 415.499, 2280.872]
p_5_C = [2478.718, -7034.501, 2280.872]

# Frame 4
p_1_4 = [4530.379, 7879.595, 1393.836]
p_2_4 = [4530.379, 3939.595, 1393.836]
p_3_4 = [2490.379, 1939.595, 1393.836]
p_4_4 = [2490.379, 419.595, 1393.836]
p_5_4 = [2490.379, -7030.405, 1393.836]

# Número de pasos para la animación
pasos = 60
espera = 0.03

# Bucle de interpolación de p_1_C a p_2_C
for i in range(pasos + 1):
    t = i / pasos

    # Interpolar posición y rotación para Frame C
    px_C = p_1_C[0] + (p_2_C[0] - p_1_C[0]) * t
    py_C = p_1_C[1] + (p_2_C[1] - p_1_C[1]) * t
    pz_C = p_1_C[2] + (p_2_C[2] - p_1_C[2]) * t

    # Interpolar posición y rotación para Frame 4
    px_4 = p_1_4[0] + (p_2_4[0] - p_1_4[0]) * t
    py_4 = p_1_4[1] + (p_2_4[1] - p_1_4[1]) * t
    pz_4 = p_1_4[2] + (p_2_4[2] - p_1_4[2]) * t

    # Aplicar las nuevas poses
    frame_C.setPose(transl(px_C, py_C, pz_C))
    frame_4.setPose(transl(px_4, py_4, pz_4))

    time.sleep(espera)

# Bucle de interpolación de p_2_C a p_3_C
for i in range(pasos + 1):
    t = i / pasos

    # Interpolar posición y rotación para Frame C
    px_C = p_2_C[0] + (p_3_C[0] - p_2_C[0]) * t
    py_C = p_2_C[1] + (p_3_C[1] - p_2_C[1]) * t
    pz_C = p_2_C[2] + (p_3_C[2] - p_2_C[2]) * t

    # Interpolar posición y rotación para Frame 4
    px_4 = p_2_4[0] + (p_3_4[0] - p_2_4[0]) * t
    py_4 = p_2_4[1] + (p_3_4[1] - p_2_4[1]) * t
    pz_4 = p_2_4[2] + (p_3_4[2] - p_2_4[2]) * t

    # Aplicar las nuevas poses
    frame_C.setPose(transl(px_C, py_C, pz_C))
    frame_4.setPose(transl(px_4, py_4, pz_4))

    time.sleep(espera)

# Bucle de interpolación de p_3_C a p_4_C
for i in range(pasos + 1):
    t = i / pasos

    # Interpolar posición y rotación para Frame C
    px_C = p_3_C[0] + (p_4_C[0] - p_3_C[0]) * t
    py_C = p_3_C[1] + (p_4_C[1] - p_3_C[1]) * t
    pz_C = p_3_C[2] + (p_4_C[2] - p_3_C[2]) * t

    # Interpolar posición y rotación para Frame 4
    px_4 = p_3_4[0] + (p_4_4[0] - p_3_4[0]) * t
    py_4 = p_3_4[1] + (p_4_4[1] - p_3_4[1]) * t
    pz_4 = p_3_4[2] + (p_4_4[2] - p_3_4[2]) * t

    # Aplicar las nuevas poses
    frame_C.setPose(transl(px_C, py_C, pz_C))
    frame_4.setPose(transl(px_4, py_4, pz_4))

    time.sleep(espera)

--- Python program MoverChopper12 ---
from robodk.robolink import *  # API de RoboDK
from robodk.robomath import *  # Funciones matemáticas
import time

# Inicializar conexión con RoboDK
RDK = Robolink()

# Obtener los frames
frame_C = RDK.Item('Frame C2', ITEM_TYPE_FRAME)
frame_4 = RDK.Item('Frame 6', ITEM_TYPE_FRAME)

if not frame_C.Valid() or not frame_4.Valid():
    raise Exception('Frames no válidos.')

# === Definir poses iniciales y finales manualmente ===

# Frame C
p_1_C = [4518.718, 7875.499, 2280.872]
p_2_C = [4518.718, 3935.499, 2280.872]
p_3_C = [2478.718, 1935.499, 2280.872]
p_4_C = [2478.718, 415.499, 2280.872]
p_5_C = [2478.718, -7034.501, 2280.872]

# Frame 4
p_1_4 = [4530.379, 7879.595, 1393.836]
p_2_4 = [4530.379, 3939.595, 1393.836]
p_3_4 = [2490.379, 1939.595, 1393.836]
p_4_4 = [2490.379, 419.595, 1393.836]
p_5_4 = [2490.379, -7030.405, 1393.836]

# Número de pasos para la animación
pasos = 60
espera = 0.03

# Bucle de interpolación de p_1_C a p_2_C
for i in range(pasos + 1):
    t = i / pasos

    # Interpolar posición y rotación para Frame C
    px_C = p_1_C[0] + (p_2_C[0] - p_1_C[0]) * t
    py_C = p_1_C[1] + (p_2_C[1] - p_1_C[1]) * t
    pz_C = p_1_C[2] + (p_2_C[2] - p_1_C[2]) * t

    # Interpolar posición y rotación para Frame 4
    px_4 = p_1_4[0] + (p_2_4[0] - p_1_4[0]) * t
    py_4 = p_1_4[1] + (p_2_4[1] - p_1_4[1]) * t
    pz_4 = p_1_4[2] + (p_2_4[2] - p_1_4[2]) * t

    # Aplicar las nuevas poses
    frame_C.setPose(transl(px_C, py_C, pz_C))
    frame_4.setPose(transl(px_4, py_4, pz_4))

    time.sleep(espera)

# Bucle de interpolación de p_2_C a p_3_C
for i in range(pasos + 1):
    t = i / pasos

    # Interpolar posición y rotación para Frame C
    px_C = p_2_C[0] + (p_3_C[0] - p_2_C[0]) * t
    py_C = p_2_C[1] + (p_3_C[1] - p_2_C[1]) * t
    pz_C = p_2_C[2] + (p_3_C[2] - p_2_C[2]) * t

    # Interpolar posición y rotación para Frame 4
    px_4 = p_2_4[0] + (p_3_4[0] - p_2_4[0]) * t
    py_4 = p_2_4[1] + (p_3_4[1] - p_2_4[1]) * t
    pz_4 = p_2_4[2] + (p_3_4[2] - p_2_4[2]) * t

    # Aplicar las nuevas poses
    frame_C.setPose(transl(px_C, py_C, pz_C))
    frame_4.setPose(transl(px_4, py_4, pz_4))

    time.sleep(espera)

# Bucle de interpolación de p_3_C a p_4_C
for i in range(pasos + 1):
    t = i / pasos

    # Interpolar posición y rotación para Frame C
    px_C = p_3_C[0] + (p_4_C[0] - p_3_C[0]) * t
    py_C = p_3_C[1] + (p_4_C[1] - p_3_C[1]) * t
    pz_C = p_3_C[2] + (p_4_C[2] - p_3_C[2]) * t

    # Interpolar posición y rotación para Frame 4
    px_4 = p_3_4[0] + (p_4_4[0] - p_3_4[0]) * t
    py_4 = p_3_4[1] + (p_4_4[1] - p_3_4[1]) * t
    pz_4 = p_3_4[2] + (p_4_4[2] - p_3_4[2]) * t

    # Aplicar las nuevas poses
    frame_C.setPose(transl(px_C, py_C, pz_C))
    frame_4.setPose(transl(px_4, py_4, pz_4))

    time.sleep(espera)

--- Python program MoverHonda21 ---
from robodk.robolink import *  # API de RoboDK
from robodk.robomath import *  # Funciones matemáticas
import time

# Inicializar conexión con RoboDK
RDK = Robolink()

# Obtener los frames
frame_H = RDK.Item('Frame H1', ITEM_TYPE_FRAME)
frame_5 = RDK.Item('Frame 5', ITEM_TYPE_FRAME)

if not frame_H.Valid() or not frame_5.Valid():
    raise Exception('Frames no válidos.')

# === Definir poses iniciales y finales manualmente ===

# Frame H
p_1_H = [448.718, 7875.499, 2280.872]
p_2_H = [448.718, 3935.499, 2280.872]
p_3_H = [2478.718, 1935.499, 2280.872]
p_4_H = [2478.718, -2534.501, 2280.872]

# Frame 5
p_1_5 = [455.915, 7880.000, 1357.578]
p_2_5 = [455.915, 3940.000, 1357.578]
p_3_5 = [2485.915, 1940.000, 1357.578]
p_4_5 = [2485.915, -2530.000, 1357.578]

# Número de pasos para la animación
pasos = 60
espera = 0.03

# Bucle de interpolación de p_1_H a p_2_H
for i in range(pasos + 1):
    t = i / pasos

    # Interpolar posición y rotación para Frame H
    px_H = p_1_H[0] + (p_2_H[0] - p_1_H[0]) * t
    py_H = p_1_H[1] + (p_2_H[1] - p_1_H[1]) * t
    pz_H = p_1_H[2] + (p_2_H[2] - p_1_H[2]) * t

    # Interpolar posición y rotación para Frame 5
    px_5 = p_1_5[0] + (p_2_5[0] - p_1_5[0]) * t
    py_5 = p_1_5[1] + (p_2_5[1] - p_1_5[1]) * t
    pz_5 = p_1_5[2] + (p_2_5[2] - p_1_5[2]) * t

    # Aplicar las nuevas poses
    frame_H.setPose(transl(px_H, py_H, pz_H))
    frame_5.setPose(transl(px_5, py_5, pz_5))

    time.sleep(espera)

# Bucle de interpolación de p_2_H a p_3_H
for i in range(pasos + 1):
    t = i / pasos

    # Interpolar posición y rotación para Frame H
    px_H = p_2_H[0] + (p_3_H[0] - p_2_H[0]) * t
    py_H = p_2_H[1] + (p_3_H[1] - p_2_H[1]) * t
    pz_H = p_2_H[2] + (p_3_H[2] - p_2_H[2]) * t

    # Interpolar posición y rotación para Frame 5
    px_5 = p_2_5[0] + (p_3_5[0] - p_2_5[0]) * t
    py_5 = p_2_5[1] + (p_3_5[1] - p_2_5[1]) * t
    pz_5 = p_2_5[2] + (p_3_5[2] - p_2_5[2]) * t

    # Aplicar las nuevas poses
    frame_H.setPose(transl(px_H, py_H, pz_H))
    frame_5.setPose(transl(px_5, py_5, pz_5))

    time.sleep(espera)

# Bucle de interpolación de p_2_H a p_3_H
for i in range(pasos + 1):
    t = i / pasos

    # Interpolar posición y rotación para Frame H
    px_H = p_3_H[0] + (p_4_H[0] - p_3_H[0]) * t
    py_H = p_3_H[1] + (p_4_H[1] - p_3_H[1]) * t
    pz_H = p_3_H[2] + (p_4_H[2] - p_3_H[2]) * t

    # Interpolar posición y rotación para Frame 5
    px_5 = p_3_5[0] + (p_4_5[0] - p_3_5[0]) * t
    py_5 = p_3_5[1] + (p_4_5[1] - p_3_5[1]) * t
    pz_5 = p_3_5[2] + (p_4_5[2] - p_3_5[2]) * t

    # Aplicar las nuevas poses
    frame_H.setPose(transl(px_H, py_H, pz_H))
    frame_5.setPose(transl(px_5, py_5, pz_5))

    time.sleep(espera)

--- Python program MoverHonda22 ---
from robodk.robolink import *  # API de RoboDK
from robodk.robomath import *  # Funciones matemáticas
import time

# Inicializar conexión con RoboDK
RDK = Robolink()

# Obtener los frames
frame_H = RDK.Item('Frame H2', ITEM_TYPE_FRAME)
frame_5 = RDK.Item('Frame 7', ITEM_TYPE_FRAME)

if not frame_H.Valid() or not frame_5.Valid():
    raise Exception('Frames no válidos.')

# === Definir poses iniciales y finales manualmente ===

# Frame H
p_1_H = [448.718, 7875.499, 2280.872]
p_2_H = [448.718, 3935.499, 2280.872]
p_3_H = [2478.718, 1935.499, 2280.872]
p_4_H = [2478.718, -2534.501, 2280.872]

# Frame 5
p_1_5 = [455.915, 7880.000, 1357.578]
p_2_5 = [455.915, 3940.000, 1357.578]
p_3_5 = [2485.915, 1940.000, 1357.578]
p_4_5 = [2485.915, -2530.000, 1357.578]

# Número de pasos para la animación
pasos = 60
espera = 0.03

# Bucle de interpolación de p_1_H a p_2_H
for i in range(pasos + 1):
    t = i / pasos

    # Interpolar posición y rotación para Frame H
    px_H = p_1_H[0] + (p_2_H[0] - p_1_H[0]) * t
    py_H = p_1_H[1] + (p_2_H[1] - p_1_H[1]) * t
    pz_H = p_1_H[2] + (p_2_H[2] - p_1_H[2]) * t

    # Interpolar posición y rotación para Frame 5
    px_5 = p_1_5[0] + (p_2_5[0] - p_1_5[0]) * t
    py_5 = p_1_5[1] + (p_2_5[1] - p_1_5[1]) * t
    pz_5 = p_1_5[2] + (p_2_5[2] - p_1_5[2]) * t

    # Aplicar las nuevas poses
    frame_H.setPose(transl(px_H, py_H, pz_H))
    frame_5.setPose(transl(px_5, py_5, pz_5))

    time.sleep(espera)

# Bucle de interpolación de p_2_H a p_3_H
for i in range(pasos + 1):
    t = i / pasos

    # Interpolar posición y rotación para Frame H
    px_H = p_2_H[0] + (p_3_H[0] - p_2_H[0]) * t
    py_H = p_2_H[1] + (p_3_H[1] - p_2_H[1]) * t
    pz_H = p_2_H[2] + (p_3_H[2] - p_2_H[2]) * t

    # Interpolar posición y rotación para Frame 5
    px_5 = p_2_5[0] + (p_3_5[0] - p_2_5[0]) * t
    py_5 = p_2_5[1] + (p_3_5[1] - p_2_5[1]) * t
    pz_5 = p_2_5[2] + (p_3_5[2] - p_2_5[2]) * t

    # Aplicar las nuevas poses
    frame_H.setPose(transl(px_H, py_H, pz_H))
    frame_5.setPose(transl(px_5, py_5, pz_5))

    time.sleep(espera)

# Bucle de interpolación de p_2_H a p_3_H
for i in range(pasos + 1):
    t = i / pasos

    # Interpolar posición y rotación para Frame H
    px_H = p_3_H[0] + (p_4_H[0] - p_3_H[0]) * t
    py_H = p_3_H[1] + (p_4_H[1] - p_3_H[1]) * t
    pz_H = p_3_H[2] + (p_4_H[2] - p_3_H[2]) * t

    # Interpolar posición y rotación para Frame 5
    px_5 = p_3_5[0] + (p_4_5[0] - p_3_5[0]) * t
    py_5 = p_3_5[1] + (p_4_5[1] - p_3_5[1]) * t
    pz_5 = p_3_5[2] + (p_4_5[2] - p_3_5[2]) * t

    # Aplicar las nuevas poses
    frame_H.setPose(transl(px_H, py_H, pz_H))
    frame_5.setPose(transl(px_5, py_5, pz_5))

    time.sleep(espera)

--- Python program MoverChopper21 ---
from robodk.robolink import *  # API de RoboDK
from robodk.robomath import *  # Funciones matemáticas
import time

# Inicializar conexión con RoboDK
RDK = Robolink()

# Obtener los frames
frame_C = RDK.Item('Frame C1', ITEM_TYPE_FRAME)
frame_4 = RDK.Item('Frame 4', ITEM_TYPE_FRAME)

if not frame_C.Valid() or not frame_4.Valid():
    raise Exception('Frames no válidos.')

# === Definir poses iniciales y finales manualmente ===

# Frame C
p_1_C = [4518.718, 7875.499, 2280.872]
p_2_C = [4518.718, 3935.499, 2280.872]
p_3_C = [2478.718, 1935.499, 2280.872]
p_4_C = [2478.718, -2534.501, 2280.872]
p_5_C = [2478.718, -7034.501, 2280.872]

# Frame 4
p_1_4 = [4530.379, 7879.595, 1393.836]
p_2_4 = [4530.379, 3939.595, 1393.836]
p_3_4 = [2490.379, 1939.595, 1393.836]
p_4_4 = [2490.379, -2530.405, 1393.836]
p_5_4 = [2490.379, -7030.405, 1393.836]

# Número de pasos para la animación
pasos = 60
espera = 0.03

# Bucle de interpolación de p_1_C a p_2_C
for i in range(pasos + 1):
    t = i / pasos

    # Interpolar posición y rotación para Frame C
    px_C = p_1_C[0] + (p_2_C[0] - p_1_C[0]) * t
    py_C = p_1_C[1] + (p_2_C[1] - p_1_C[1]) * t
    pz_C = p_1_C[2] + (p_2_C[2] - p_1_C[2]) * t

    # Interpolar posición y rotación para Frame 4
    px_4 = p_1_4[0] + (p_2_4[0] - p_1_4[0]) * t
    py_4 = p_1_4[1] + (p_2_4[1] - p_1_4[1]) * t
    pz_4 = p_1_4[2] + (p_2_4[2] - p_1_4[2]) * t

    # Aplicar las nuevas poses
    frame_C.setPose(transl(px_C, py_C, pz_C))
    frame_4.setPose(transl(px_4, py_4, pz_4))

    time.sleep(espera)

# Bucle de interpolación de p_2_C a p_3_C
for i in range(pasos + 1):
    t = i / pasos

    # Interpolar posición y rotación para Frame C
    px_C = p_2_C[0] + (p_3_C[0] - p_2_C[0]) * t
    py_C = p_2_C[1] + (p_3_C[1] - p_2_C[1]) * t
    pz_C = p_2_C[2] + (p_3_C[2] - p_2_C[2]) * t

    # Interpolar posición y rotación para Frame 4
    px_4 = p_2_4[0] + (p_3_4[0] - p_2_4[0]) * t
    py_4 = p_2_4[1] + (p_3_4[1] - p_2_4[1]) * t
    pz_4 = p_2_4[2] + (p_3_4[2] - p_2_4[2]) * t

    # Aplicar las nuevas poses
    frame_C.setPose(transl(px_C, py_C, pz_C))
    frame_4.setPose(transl(px_4, py_4, pz_4))

    time.sleep(espera)

# Bucle de interpolación de p_3_C a p_4_C
for i in range(pasos + 1):
    t = i / pasos

    # Interpolar posición y rotación para Frame C
    px_C = p_3_C[0] + (p_4_C[0] - p_3_C[0]) * t
    py_C = p_3_C[1] + (p_4_C[1] - p_3_C[1]) * t
    pz_C = p_3_C[2] + (p_4_C[2] - p_3_C[2]) * t

    # Interpolar posición y rotación para Frame 4
    px_4 = p_3_4[0] + (p_4_4[0] - p_3_4[0]) * t
    py_4 = p_3_4[1] + (p_4_4[1] - p_3_4[1]) * t
    pz_4 = p_3_4[2] + (p_4_4[2] - p_3_4[2]) * t

    # Aplicar las nuevas poses
    frame_C.setPose(transl(px_C, py_C, pz_C))
    frame_4.setPose(transl(px_4, py_4, pz_4))

    time.sleep(espera)

--- Python program MoverChopper22 ---
from robodk.robolink import *  # API de RoboDK
from robodk.robomath import *  # Funciones matemáticas
import time

# Inicializar conexión con RoboDK
RDK = Robolink()

# Obtener los frames
frame_C = RDK.Item('Frame C2', ITEM_TYPE_FRAME)
frame_4 = RDK.Item('Frame 6', ITEM_TYPE_FRAME)

if not frame_C.Valid() or not frame_4.Valid():
    raise Exception('Frames no válidos.')

# === Definir poses iniciales y finales manualmente ===

# Frame C
p_1_C = [4518.718, 7875.499, 2280.872]
p_2_C = [4518.718, 3935.499, 2280.872]
p_3_C = [2478.718, 1935.499, 2280.872]
p_4_C = [2478.718, -2534.501, 2280.872]
p_5_C = [2478.718, -7034.501, 2280.872]

# Frame 4
p_1_4 = [4530.379, 7879.595, 1393.836]
p_2_4 = [4530.379, 3939.595, 1393.836]
p_3_4 = [2490.379, 1939.595, 1393.836]
p_4_4 = [2490.379, -2530.405, 1393.836]
p_5_4 = [2490.379, -7030.405, 1393.836]

# Número de pasos para la animación
pasos = 60
espera = 0.03

# Bucle de interpolación de p_1_C a p_2_C
for i in range(pasos + 1):
    t = i / pasos

    # Interpolar posición y rotación para Frame C
    px_C = p_1_C[0] + (p_2_C[0] - p_1_C[0]) * t
    py_C = p_1_C[1] + (p_2_C[1] - p_1_C[1]) * t
    pz_C = p_1_C[2] + (p_2_C[2] - p_1_C[2]) * t

    # Interpolar posición y rotación para Frame 4
    px_4 = p_1_4[0] + (p_2_4[0] - p_1_4[0]) * t
    py_4 = p_1_4[1] + (p_2_4[1] - p_1_4[1]) * t
    pz_4 = p_1_4[2] + (p_2_4[2] - p_1_4[2]) * t

    # Aplicar las nuevas poses
    frame_C.setPose(transl(px_C, py_C, pz_C))
    frame_4.setPose(transl(px_4, py_4, pz_4))

    time.sleep(espera)

# Bucle de interpolación de p_2_C a p_3_C
for i in range(pasos + 1):
    t = i / pasos

    # Interpolar posición y rotación para Frame C
    px_C = p_2_C[0] + (p_3_C[0] - p_2_C[0]) * t
    py_C = p_2_C[1] + (p_3_C[1] - p_2_C[1]) * t
    pz_C = p_2_C[2] + (p_3_C[2] - p_2_C[2]) * t

    # Interpolar posición y rotación para Frame 4
    px_4 = p_2_4[0] + (p_3_4[0] - p_2_4[0]) * t
    py_4 = p_2_4[1] + (p_3_4[1] - p_2_4[1]) * t
    pz_4 = p_2_4[2] + (p_3_4[2] - p_2_4[2]) * t

    # Aplicar las nuevas poses
    frame_C.setPose(transl(px_C, py_C, pz_C))
    frame_4.setPose(transl(px_4, py_4, pz_4))

    time.sleep(espera)

# Bucle de interpolación de p_3_C a p_4_C
for i in range(pasos + 1):
    t = i / pasos

    # Interpolar posición y rotación para Frame C
    px_C = p_3_C[0] + (p_4_C[0] - p_3_C[0]) * t
    py_C = p_3_C[1] + (p_4_C[1] - p_3_C[1]) * t
    pz_C = p_3_C[2] + (p_4_C[2] - p_3_C[2]) * t

    # Interpolar posición y rotación para Frame 4
    px_4 = p_3_4[0] + (p_4_4[0] - p_3_4[0]) * t
    py_4 = p_3_4[1] + (p_4_4[1] - p_3_4[1]) * t
    pz_4 = p_3_4[2] + (p_4_4[2] - p_3_4[2]) * t

    # Aplicar las nuevas poses
    frame_C.setPose(transl(px_C, py_C, pz_C))
    frame_4.setPose(transl(px_4, py_4, pz_4))

    time.sleep(espera)

--- Python program MoverChopper11Final ---
from robodk.robolink import *  # API de RoboDK
from robodk.robomath import *  # Funciones matemáticas
import time

# Inicializar conexión con RoboDK
RDK = Robolink()

# Obtener los frames
frame_C = RDK.Item('Frame C1', ITEM_TYPE_FRAME)
frame_4 = RDK.Item('Frame 4', ITEM_TYPE_FRAME)

# Obtener el objeto
obj = RDK.Item('Chopper Frame AP203 1', ITEM_TYPE_OBJECT)

if not frame_C.Valid() or not frame_4.Valid():
    raise Exception('Frames no válidos.')

# Frame C
p_4_C = [2478.718, 415.499, 2280.872]
p_5_C = [2478.718, -7034.501, 2280.872]

# Frame 4
p_4_4 = [2490.379, 419.595, 1393.836]
p_5_4 = [2490.379, -7030.405, 1393.836]

# Número de pasos para la animación
pasos = 60
espera = 0.03

# Bucle de interpolación de p_4_C a p_5_C
for i in range(pasos + 1):
    t = i / pasos

    # Interpolar posición y rotación para Frame C
    px_C = p_4_C[0] + (p_5_C[0] - p_4_C[0]) * t
    py_C = p_4_C[1] + (p_5_C[1] - p_4_C[1]) * t
    pz_C = p_4_C[2] + (p_5_C[2] - p_4_C[2]) * t

    # Interpolar posición y rotación para Frame 4
    px_4 = p_4_4[0] + (p_5_4[0] - p_4_4[0]) * t
    py_4 = p_4_4[1] + (p_5_4[1] - p_4_4[1]) * t
    pz_4 = p_4_4[2] + (p_5_4[2] - p_4_4[2]) * t

    # Aplicar las nuevas poses
    frame_C.setPose(transl(px_C, py_C, pz_C))
    frame_4.setPose(transl(px_4, py_4, pz_4))

    time.sleep(espera)

obj.setColor([0.9, 0.9, 0.9, 1.0])

--- Python program MoverChopper12Final ---
from robodk.robolink import *  # API de RoboDK
from robodk.robomath import *  # Funciones matemáticas
import time

# Inicializar conexión con RoboDK
RDK = Robolink()

# Obtener los frames
frame_C = RDK.Item('Frame C2', ITEM_TYPE_FRAME)
frame_4 = RDK.Item('Frame 6', ITEM_TYPE_FRAME)

# Obtener el objeto
obj = RDK.Item('Chopper Frame AP203 2', ITEM_TYPE_OBJECT)

if not frame_C.Valid() or not frame_4.Valid():
    raise Exception('Frames no válidos.')

# Frame C
p_4_C = [2478.718, 415.499, 2280.872]
p_5_C = [2478.718, -7034.501, 2280.872]

# Frame 4
p_4_4 = [2490.379, 419.595, 1393.836]
p_5_4 = [2490.379, -7030.405, 1393.836]

# Número de pasos para la animación
pasos = 60
espera = 0.03

# Bucle de interpolación de p_4_C a p_5_C
for i in range(pasos + 1):
    t = i / pasos

    # Interpolar posición y rotación para Frame C
    px_C = p_4_C[0] + (p_5_C[0] - p_4_C[0]) * t
    py_C = p_4_C[1] + (p_5_C[1] - p_4_C[1]) * t
    pz_C = p_4_C[2] + (p_5_C[2] - p_4_C[2]) * t

    # Interpolar posición y rotación para Frame 4
    px_4 = p_4_4[0] + (p_5_4[0] - p_4_4[0]) * t
    py_4 = p_4_4[1] + (p_5_4[1] - p_4_4[1]) * t
    pz_4 = p_4_4[2] + (p_5_4[2] - p_4_4[2]) * t

    # Aplicar las nuevas poses
    frame_C.setPose(transl(px_C, py_C, pz_C))
    frame_4.setPose(transl(px_4, py_4, pz_4))

    time.sleep(espera)

obj.setColor([0.9, 0.9, 0.9, 1.0])

--- Python program MoverHonda11Final ---
from robodk.robolink import *  # API de RoboDK
from robodk.robomath import *  # Funciones matemáticas
import time
import math

# Inicializar conexión con RoboDK
RDK = Robolink()

# Obtener los frames
frame_H = RDK.Item('Frame H1', ITEM_TYPE_FRAME)
frame_5 = RDK.Item('Frame 5', ITEM_TYPE_FRAME)

# Obtener el objeto
obj = RDK.Item('Frame cb 750 1', ITEM_TYPE_OBJECT)

if not frame_H.Valid() or not frame_5.Valid():
    raise Exception('Frames no válidos.')

# Frame H
p_4_H = [2478.718, 415.499, 2280.872]
p_5_H = [2478.718, -7034.501, 2280.872]

# Frame 5
p_4_5 = [2485.915, 420.000, 1357.578]
p_5_5 = [2485.915, -7030.000, 1357.578]

# Número de pasos para la animación
pasos = 60
espera = 0.03

# Bucle de interpolación de p_4_H a p_5_H
for i in range(pasos + 1):
    t = i / pasos

    # Interpolar posición y rotación para Frame H
    px_H = p_4_H[0] + (p_5_H[0] - p_4_H[0]) * t
    py_H = p_4_H[1] + (p_5_H[1] - p_4_H[1]) * t
    pz_H = p_4_H[2] + (p_5_H[2] - p_4_H[2]) * t

    # Interpolar posición y rotación para Frame 5
    px_5 = p_4_5[0] + (p_5_5[0] - p_4_5[0]) * t
    py_5 = p_4_5[1] + (p_5_5[1] - p_4_5[1]) * t
    pz_5 = p_4_5[2] + (p_5_5[2] - p_4_5[2]) * t

    # Aplicar las nuevas poses
    frame_H.setPose(transl(px_H, py_H, pz_H))
    frame_5.setPose(transl(px_5, py_5, pz_5))

    time.sleep(espera)

obj.setColor([0.9, 0.9, 0.9, 1.0])

--- Python program MoverHonda12Final ---
from robodk.robolink import *  # API de RoboDK
from robodk.robomath import *  # Funciones matemáticas
import time
import math

# Inicializar conexión con RoboDK
RDK = Robolink()

# Obtener los frames
frame_H = RDK.Item('Frame H2', ITEM_TYPE_FRAME)
frame_5 = RDK.Item('Frame 7', ITEM_TYPE_FRAME)

# Obtener el objeto
obj = RDK.Item('Frame cb 750 2', ITEM_TYPE_OBJECT)

if not frame_H.Valid() or not frame_5.Valid():
    raise Exception('Frames no válidos.')

# Frame H
p_4_H = [2478.718, 415.499, 2280.872]
p_5_H = [2478.718, -7034.501, 2280.872]

# Frame 5
p_4_5 = [2485.915, 420.000, 1357.578]
p_5_5 = [2485.915, -7030.000, 1357.578]

# Número de pasos para la animación
pasos = 60
espera = 0.03

# Bucle de interpolación de p_4_H a p_5_H
for i in range(pasos + 1):
    t = i / pasos

    # Interpolar posición y rotación para Frame H
    px_H = p_4_H[0] + (p_5_H[0] - p_4_H[0]) * t
    py_H = p_4_H[1] + (p_5_H[1] - p_4_H[1]) * t
    pz_H = p_4_H[2] + (p_5_H[2] - p_4_H[2]) * t

    # Interpolar posición y rotación para Frame 5
    px_5 = p_4_5[0] + (p_5_5[0] - p_4_5[0]) * t
    py_5 = p_4_5[1] + (p_5_5[1] - p_4_5[1]) * t
    pz_5 = p_4_5[2] + (p_5_5[2] - p_4_5[2]) * t

    # Aplicar las nuevas poses
    frame_H.setPose(transl(px_H, py_H, pz_H))
    frame_5.setPose(transl(px_5, py_5, pz_5))

    time.sleep(espera)

obj.setColor([0.9, 0.9, 0.9, 1.0])

--- Python program MoverChopper21Final ---
from robodk.robolink import *  # API de RoboDK
from robodk.robomath import *  # Funciones matemáticas
import time

# Inicializar conexión con RoboDK
RDK = Robolink()

# Obtener los frames
frame_C = RDK.Item('Frame C1', ITEM_TYPE_FRAME)
frame_4 = RDK.Item('Frame 4', ITEM_TYPE_FRAME)

# Obtener el objeto
obj = RDK.Item('Chopper Frame AP203 1', ITEM_TYPE_OBJECT)

if not frame_C.Valid() or not frame_4.Valid():
    raise Exception('Frames no válidos.')

# Frame C
p_4_C = [2478.718, -2534.501, 2280.872]
p_5_C = [2478.718, -7034.501, 2280.872]

# Frame 4
p_4_4 = [2490.379, -2530.405, 1393.836]
p_5_4 = [2490.379, -7030.405, 1393.836]

# Número de pasos para la animación
pasos = 60
espera = 0.03

# Bucle de interpolación de p_4_C a p_5_C
for i in range(pasos + 1):
    t = i / pasos

    # Interpolar posición y rotación para Frame C
    px_C = p_4_C[0] + (p_5_C[0] - p_4_C[0]) * t
    py_C = p_4_C[1] + (p_5_C[1] - p_4_C[1]) * t
    pz_C = p_4_C[2] + (p_5_C[2] - p_4_C[2]) * t

    # Interpolar posición y rotación para Frame 4
    px_4 = p_4_4[0] + (p_5_4[0] - p_4_4[0]) * t
    py_4 = p_4_4[1] + (p_5_4[1] - p_4_4[1]) * t
    pz_4 = p_4_4[2] + (p_5_4[2] - p_4_4[2]) * t

    # Aplicar las nuevas poses
    frame_C.setPose(transl(px_C, py_C, pz_C))
    frame_4.setPose(transl(px_4, py_4, pz_4))

    time.sleep(espera)

obj.setColor([0.9, 0.9, 0.9, 1.0])

--- Python program MoverChopper22Final ---
from robodk.robolink import *  # API de RoboDK
from robodk.robomath import *  # Funciones matemáticas
import time

# Inicializar conexión con RoboDK
RDK = Robolink()

# Obtener los frames
frame_C = RDK.Item('Frame C2', ITEM_TYPE_FRAME)
frame_4 = RDK.Item('Frame 6', ITEM_TYPE_FRAME)

# Obtener el objeto
obj = RDK.Item('Chopper Frame AP203 2', ITEM_TYPE_OBJECT)

if not frame_C.Valid() or not frame_4.Valid():
    raise Exception('Frames no válidos.')

# Frame C
p_4_C = [2478.718, -2534.501, 2280.872]
p_5_C = [2478.718, -7034.501, 2280.872]

# Frame 4
p_4_4 = [2490.379, -2530.405, 1393.836]
p_5_4 = [2490.379, -7030.405, 1393.836]

# Número de pasos para la animación
pasos = 60
espera = 0.03

# Bucle de interpolación de p_4_C a p_5_C
for i in range(pasos + 1):
    t = i / pasos

    # Interpolar posición y rotación para Frame C
    px_C = p_4_C[0] + (p_5_C[0] - p_4_C[0]) * t
    py_C = p_4_C[1] + (p_5_C[1] - p_4_C[1]) * t
    pz_C = p_4_C[2] + (p_5_C[2] - p_4_C[2]) * t

    # Interpolar posición y rotación para Frame 4
    px_4 = p_4_4[0] + (p_5_4[0] - p_4_4[0]) * t
    py_4 = p_4_4[1] + (p_5_4[1] - p_4_4[1]) * t
    pz_4 = p_4_4[2] + (p_5_4[2] - p_4_4[2]) * t

    # Aplicar las nuevas poses
    frame_C.setPose(transl(px_C, py_C, pz_C))
    frame_4.setPose(transl(px_4, py_4, pz_4))

    time.sleep(espera)

obj.setColor([0.9, 0.9, 0.9, 1.0])

--- Python program MoverHonda21Final ---
from robodk.robolink import *  # API de RoboDK
from robodk.robomath import *  # Funciones matemáticas
import time

# Inicializar conexión con RoboDK
RDK = Robolink()

# Obtener los frames
frame_H = RDK.Item('Frame H1', ITEM_TYPE_FRAME)
frame_5 = RDK.Item('Frame 5', ITEM_TYPE_FRAME)

# Obtener el objeto
obj = RDK.Item('Frame cb 750 1', ITEM_TYPE_OBJECT)

if not frame_H.Valid() or not frame_5.Valid():
    raise Exception('Frames no válidos.')

# Frame H
p_4_H = [2478.718, -2534.501, 2280.872]
p_5_H = [2478.718, -7034.501, 2280.872]

# Frame 5
p_4_5 = [2485.915, -2530.000, 1357.578]
p_5_5 = [2485.915, -7030.000, 1357.578]

# Número de pasos para la animación
pasos = 60
espera = 0.03

# Bucle de interpolación de p_4_H a p_5_H
for i in range(pasos + 1):
    t = i / pasos

    # Interpolar posición y rotación para Frame H
    px_H = p_4_H[0] + (p_5_H[0] - p_4_H[0]) * t
    py_H = p_4_H[1] + (p_5_H[1] - p_4_H[1]) * t
    pz_H = p_4_H[2] + (p_5_H[2] - p_4_H[2]) * t

    # Interpolar posición y rotación para Frame 5
    px_5 = p_4_5[0] + (p_5_5[0] - p_4_5[0]) * t
    py_5 = p_4_5[1] + (p_5_5[1] - p_4_5[1]) * t
    pz_5 = p_4_5[2] + (p_5_5[2] - p_4_5[2]) * t

    # Aplicar las nuevas poses
    frame_H.setPose(transl(px_H, py_H, pz_H))
    frame_5.setPose(transl(px_5, py_5, pz_5))

    time.sleep(espera)

obj.setColor([0.9, 0.9, 0.9, 1.0])

--- Python program MoverHonda22Final ---
from robodk.robolink import *  # API de RoboDK
from robodk.robomath import *  # Funciones matemáticas
import time

# Inicializar conexión con RoboDK
RDK = Robolink()

# Obtener los frames
frame_H = RDK.Item('Frame H2', ITEM_TYPE_FRAME)
frame_5 = RDK.Item('Frame 7', ITEM_TYPE_FRAME)

# Obtener el objeto
obj = RDK.Item('Frame cb 750 2', ITEM_TYPE_OBJECT)

if not frame_H.Valid() or not frame_5.Valid():
    raise Exception('Frames no válidos.')

# Frame H
p_4_H = [2478.718, -2534.501, 2280.872]
p_5_H = [2478.718, -7034.501, 2280.872]

# Frame 5
p_4_5 = [2485.915, -2530.000, 1357.578]
p_5_5 = [2485.915, -7030.000, 1357.578]

# Número de pasos para la animación
pasos = 60
espera = 0.03

# Bucle de interpolación de p_4_H a p_5_H
for i in range(pasos + 1):
    t = i / pasos

    # Interpolar posición y rotación para Frame H
    px_H = p_4_H[0] + (p_5_H[0] - p_4_H[0]) * t
    py_H = p_4_H[1] + (p_5_H[1] - p_4_H[1]) * t
    pz_H = p_4_H[2] + (p_5_H[2] - p_4_H[2]) * t

    # Interpolar posición y rotación para Frame 5
    px_5 = p_4_5[0] + (p_5_5[0] - p_4_5[0]) * t
    py_5 = p_4_5[1] + (p_5_5[1] - p_4_5[1]) * t
    pz_5 = p_4_5[2] + (p_5_5[2] - p_4_5[2]) * t

    # Aplicar las nuevas poses
    frame_H.setPose(transl(px_H, py_H, pz_H))
    frame_5.setPose(transl(px_5, py_5, pz_5))

    time.sleep(espera)

obj.setColor([0.9, 0.9, 0.9, 1.0])

--- Python program Reset ---
from robodk.robolink import *  # API de RoboDK
from robodk.robomath import *  # Funciones matemáticas
import time
import math

# Inicializar conexión con RoboDK
RDK = Robolink()

# Color neutro inicial
color_inicial = [0.9, 0.9, 0.9, 1.0]

# Obtener los frames
frame_H1 = RDK.Item('Frame H1', ITEM_TYPE_FRAME)
frame_5 = RDK.Item('Frame 5', ITEM_TYPE_FRAME)
honda1 = RDK.Item('Frame cb 750 1', ITEM_TYPE_OBJECT)

if not frame_H1.Valid() or not frame_5.Valid():
    raise Exception('Frames no válidos.')

frame_H2 = RDK.Item('Frame H2', ITEM_TYPE_FRAME)
frame_7 = RDK.Item('Frame 7', ITEM_TYPE_FRAME)
honda2 = RDK.Item('Frame cb 750 2', ITEM_TYPE_OBJECT)

if not frame_H2.Valid() or not frame_7.Valid():
    raise Exception('Frames no válidos.')

frame_C1 = RDK.Item('Frame C1', ITEM_TYPE_FRAME)
frame_4 = RDK.Item('Frame 4', ITEM_TYPE_FRAME)
chopper1 = RDK.Item('Chopper Frame AP203 1', ITEM_TYPE_OBJECT)

if not frame_C1.Valid() or not frame_4.Valid():
    raise Exception('Frames no válidos.')

frame_C2 = RDK.Item('Frame C2', ITEM_TYPE_FRAME)
frame_6 = RDK.Item('Frame 6', ITEM_TYPE_FRAME)
chopper2 = RDK.Item('Chopper Frame AP203 2', ITEM_TYPE_OBJECT)

if not frame_C2.Valid() or not frame_6.Valid():
    raise Exception('Frames no válidos.')

# === Definir poses iniciales y finales manualmente ===

# Frame C1
p_1_C1 = [4518.718, 7875.499, 2280.872]

# Frame 4
p_1_4 = [4530.379, 7879.595, 1393.836]

# Frame C2
p_1_C2 = [4518.718, 7875.499, 2280.872]

# Frame 6
p_1_6 = [4530.379, 7879.595, 1393.836]

# Frame H1
p_1_H1 = [448.718, 7875.499, 2280.872]

# Frame 5
p_1_5 = [455.915, 7880.000, 1357.578]

# Frame H2
p_1_H2 = [448.718, 7875.499, 2280.872]

# Frame 7
p_1_7 = [455.915, 7880.000, 1357.578]

# Aplicar las nuevas poses
frame_H1.setPose(transl(p_1_H1))
frame_5.setPose(transl(p_1_5))
honda1.setColor(color_inicial)

frame_H2.setPose(transl(p_1_H2))
frame_7.setPose(transl(p_1_7))
honda2.setColor(color_inicial)

frame_C1.setPose(transl(p_1_C1))
frame_4.setPose(transl(p_1_4))
chopper1.setColor(color_inicial)

frame_C2.setPose(transl(p_1_C2))
frame_6.setPose(transl(p_1_6))
chopper2.setColor(color_inicial)

--- program Honda1Robot1 (robot ABB IRB 580/12S 2) ---
  Llamar MoverHonda11
  Llamar Honda11
  Llamar MoverHonda11Final
  Set Robot1Operando=0

--- program Honda2Robot1 (robot ABB IRB 580/12S 2) ---
  Llamar MoverHonda12
  Llamar Honda12
  Llamar MoverHonda12Final
  Set Robot1Operando=0

--- program Honda1Robot2 (robot ABB IRB 580/12S 2) ---
  Llamar MoverHonda21
  Llamar Honda21
  Llamar MoverHonda21Final
  Set Robot2Operando=0

--- program Chopper1Robot1 (robot ABB IRB 580/12S 2) ---
  Llamar MoverChopper11
  Llamar Chopper11
  Llamar MoverChopper11Final
  Set Robot1Operando=0

--- program Chopper2Robot1 (robot ABB IRB 580/12S 2) ---
  Llamar MoverChopper12
  Llamar Chopper12
  Llamar MoverChopper12Final
  Set Robot1Operando=0

--- program Chopper1Robot2 (robot ABB IRB 580/12S 2) ---
  Llamar MoverChopper21
  Llamar Chopper21
  Llamar MoverChopper21Final
  Set Robot2Operando=0

--- program Reset (robot ABB IRB 580/12S 2) ---
  Llamar Reset
